KUKA KRL program: RoboSyncPrint.src, RoboSyncPrint.dat

--- RoboSyncPrint.src ---
&ACCESS RVO3
&REL 16
&PARAM DISKPATH = KRC:\R1\TP\CNCRobotics\CEAD
DEF RoboSyncPrint( )
;************************************************
;     NextState Automation Ltd
;     www.nextstateautomation.co.uk
;************************************************
;     Contact: helpdesk@nextstateautomation.co.uk
;     Date: 14/09/26
;     Version: 0.1.1
;     Module : RoboSyncPrint
;     Purpose: Stepper drive commands and parameters for the RoboSync Hub
;************************************************
END

GLOBAL DEF StartPrint()
;------------------------------------------------
; Name    : StartPrint
; Purpose : Write one stepper drive parameter
; Params  : -
; Returns : -
; Notes   : Controls the Heatzones and Stepper before printing
;
;------------------------------------------------

rFilamentOD = 2.85
rLayerHeight = 0.5
rLayerWidth = 0.5

rExtrusionConstant = 1.0

SetExtruderHeatZones(180.0, 180.0)


WaitForExtruderTemps()

bSpsControl = TRUE
bEnableRetract = FALSE
bEnableStepper = TRUE
WAIT FOR stepperState
bExtrude = FALSE
WAIT FOR stepperState == #RUNNNING

END

GLOBAL DEF FinishPrint()
;------------------------------------------------
; Name    : StartPrint
; Purpose : Write one stepper drive parameter
; Params  : -
; Returns : -
; Notes   : Controls the Heatzones and Stepper before printing
;
;------------------------------------------------

SetExtruderHeatZones(0.0, 0.0)

WaitForExtruderTemps()

bSpsControl = TRUE
bEnableRetract = FALSE
bExtrude = FALSE
bEnableStepper = FALSE


WAIT FOR stepperState == #RUNNNING

END

--- RoboSyncPrint.dat ---
&ACCESS RVO3
&REL 16
&PARAM DISKPATH = KRC:\R1\TP\CNCRobotics\CEAD
DEFDAT  RoboSyncPrint PUBLIC
;************************************************
;     NextState Automation Ltd
;     www.nextstateautomation.co.uk
;************************************************
;     Contact: helpdesk@nextstate.co.uk
;     Date: 14/09/26
;     Version: 0.1.1
;************************************************

GLOBAL CONST INT RESET_ALARM_CODE=186
GLOBAL CONST INT ENABLE_DRIVE=159
GLOBAL CONST INT DISABLE_DRIVE=158
GLOBAL CONST INT COMMENCE_JOGGING=150
GLOBAL CONST INT STOP_JOGGING=216
GLOBAL CONST INT MOVE_RELATIVE_DISTANCE=102
GLOBAL CONST INT MOVE_ABSOLUTE_DISTANCE=103
GLOBAL CONST INT FAST_STOP_MOVE=225
GLOBAL CONST INT STOP_MOVE=226
GLOBAL CONST INT SET_POSITION = 165

GLOBAL ENUM ENUM_STEPPER_PARAM CURRENT,IDLE_CURRENT,PULSE_PER_REV,JOG_SPEED,JOG_ACCEL,JOG_DECEL,SPEED,ACCEL,DECEL,DISTANCE,SET_POSITION

ENDDAT
